PROGRAM MAIN
VAR
	fbNewEngine			: FB_NewEngine;	
END_VAR

fbNewEngine.Start(1, 7.5);

END_PROGRAM

(* stored: Version 1.1.0.1, ProductVersion 3.1.4020.12
   POU MAIN: Id {956a2d5c-6bee-4359-b4e8-bbb283d0e9fa}, SpecialFunc None *)
